(*
A definition of a struct.
*)
TYPE AutoStruct :
STRUCT
    someDouble          : LREAL;        // Use to store a number
    someBoolean         : BOOL;         // Use as a flag
END_STRUCT
END_TYPE

(* stored: Version 1.1.0.1, ProductVersion 3.1.4024.11
   DUT AutoStruct: Id {1c2a330d-7850-4ffb-ad1e-06aa955e96eb} *)
